{attribute 'GeneratedUsingTerminal: AX8108-0100-0101-0101'}
{attribute addProperty BoxType "AX8108-0100-0101-0101"}
{attribute addProperty Id "Safe_Logic_StateUSINT1Cycle_CounterUSINT1"}
{attribute addProperty CRC "331147839"}
{attribute addProperty Size "2"}
TYPE FSOE_13BCEA3F :
STRUCT
	{attribute addProperty Name "Safe_Logic_State"}
	Safe_Logic_State : USINT;
	{attribute addProperty Name "Cycle_Counter"}
	Cycle_Counter : USINT;
END_STRUCT
END_TYPE

(* stored: Version 1.2.0.0, ProductVersion 3.1.4024.9
   DUT FSOE_13BCEA3F: Id {8a5e8272-3c10-4ebc-bef3-5ab9dfdda21a} *)
